// TwinCAT 3 PLC project Testing
// ProgramVersion: 3.1.4026.13
// libraries:
//   Tc2_Standard, * (Beckhoff Automation GmbH)
//   Tc2_System, * (Beckhoff Automation GmbH)
//   Tc3_Component, * (Zerlauth)
//   Tc3_Module, * (Beckhoff Automation GmbH)
//   Tc3_UnitTest, * (Zerlauth)
// project tree:
//   / PlcTask.TcTTO
//   POUs/ MAIN.TcPOU
//   Tests/ FB_ListComponentTests.TcPOU, FB_ListObjectTests.TcPOU, FB_ListStringTests.TcPOU, FB_MembersTests.TcPOU, FB_ComponentTests.TcPOU
// (motion and I/O tree: see PLC project development)
// real-time tasks:
//   TASK PlcTask: cycle T#500ms, priority 21, ADS port 351
//   TASK UnitTestTask: cycle T#1ms, priority 1, ADS port 350
// variable links:

CONFIGURATION Testing
    RESOURCE PLC ON TwinCAT3
        TASK PlcTask(INTERVAL := T#500ms, PRIORITY := 21);
        PROGRAM MAIN WITH PlcTask : MAIN;
    END_RESOURCE
END_CONFIGURATION

// ---- POUs/MAIN.TcPOU
PROGRAM MAIN
VAR
	bInitialise: 			BOOL:= TRUE;
	bExecute: 				BOOL;
	fbTestsuites:			FB_Testsuites;
	fbListObject:			FB_ListObjectTests;
	fbListComponent:		FB_ListComponentTests;
	fbListString:			FB_ListStringTests;
	fbMembers:				FB_MembersTests;
	fbComponentTests:		FB_ComponentTests;
END_VAR

IF bInitialise THEN
	bInitialise:= False;
	fbTestsuites.M_Add(fbListObject.fbTestsuite);
	fbTestsuites.M_Add(fbListComponent.fbTestsuite);
	fbTestsuites.M_Add(fbListString.fbTestsuite);
	fbTestsuites.M_Add(fbMembers.fbTestsuite);
	fbTestsuites.M_Add(fbComponentTests.fbTestsuite);
	fbTestsuites.P_Options.sFilePathName:= 'C:\report.xml';
END_IF

IF bExecute THEN
	bExecute:= fbTestsuites.M_Request(E_Base.Execute);
END_IF

fbTestsuites();


fbListObject();
fbListComponent();
fbListString();
fbMembers();
fbComponentTests();

END_PROGRAM

// ---- Tests/FB_ListObjectTests.TcPOU
FUNCTION_BLOCK FB_ListObjectTests EXTENDS 
VAR_INPUT
END_VAR
VAR_OUTPUT
	fbTestsuite:			FB_Testsuite;
END_VAR
VAR
	fbList:					Tc3_Component.FB_ListObject;
	fbObject:				Tc3_Component.FB_Object;
	iObject:				Tc3_Component.I_Object:= fbObject;
END_VAR

fbTestsuite.P_Property.M_Add('object', 'FB_ListObject');
fbTestsuite.P_Property.M_Add('name', 'Peter Zerlauth');

fbTestsuite();

CASE fbTestsuite.P_Testcase OF
	
	E_Testcase.Start:
		fbTestsuite.P_Assert.M_Equals_DINT(fbList.P_Length, 0, 'P_Length');
		fbTestsuite.M_Testcase('FB_ListObject', T#2S, 'fbList.P_Length', '', 10);	
		
	10:
		fbTestsuite.P_Assert.M_Equals_BOOL(fbList.M_Add(fbObject), TRUE, 'M_Add(fbObject)');
		fbTestsuite.M_Testcase('FB_ListObject', T#2S, 'fbList.M_Add(fbObject)', '', 20);
		
	20:
		fbTestsuite.P_Assert.M_Equals_DINT(fbList.P_Length, 1, 'P_Length');
		fbTestsuite.M_Testcase('FB_ListObject', T#2S, 'fbList.P_Length', '', 30);		
		
	30:
		fbTestsuite.P_Assert.M_Equals_DINT(fbList.M_Find(fbObject), 0, 'M_Find');
		fbTestsuite.M_Testcase('FB_ListObject', T#2S, 'fbList.M_Find(fbObject)', '', 40);
		
	40:

		fbTestsuite.P_Assert.M_Equals_BOOL(TRUE, __QUERYINTERFACE(fbList.M_Index(0), iObject), 'M_Index');
		fbTestsuite.M_Testcase('FB_ListObject', T#2S, 'fbList.M_Index(1)', '', 50);
		
	50:
		fbTestsuite.P_Assert.M_Equals_BOOL(fbList.M_Remove(fbObject), TRUE, 'M_Remove');
		fbTestsuite.M_Testcase('FB_ListObject', T#2S, 'fbList.M_Remove(fbObject', '', 60);		

	60:
		fbTestsuite.P_Assert.M_Equals_DINT(fbList.P_Length, 0, 'P_Length');
		fbTestsuite.M_Testcase('FB_ListObject', T#2S, 'fbList.P_Length', '', 70);
		
	70:
		fbTestsuite.P_Assert.M_Equals_BOOL(fbList.M_Add(fbObject), TRUE, 'M_Add(fbObject)');
		fbTestsuite.M_Testcase('FB_ListObject', T#2S, 'fbList.M_Add(fbObject)', '', 80);

	80:
		fbTestsuite.P_Assert.M_Equals_DINT(fbList.P_Length, 1, 'P_Length');
		fbTestsuite.M_Testcase('FB_ListObject', T#2S, 'fbList.P_Length', '', 90);
		
	90:
		fbTestsuite.P_Assert.M_Equals_BOOL(fbList.M_Clear(), TRUE, 'M_Clear()');
		fbTestsuite.M_Testcase('FB_ListObject', T#2S, 'fbList.M_Clear()', '', 100);		
	
	100:
		fbTestsuite.P_Assert.M_Equals_DINT(fbList.P_Length, 0, 'P_Length');
		fbTestsuite.M_Testcase('FB_ListObject', T#2S, 'fbList.P_Length', '', E_Testcase.Done);
		
	E_Testcase.Done:
		;
END_CASE

END_FUNCTION_BLOCK

// ---- Tests/FB_ListComponentTests.TcPOU
FUNCTION_BLOCK FB_ListComponentTests EXTENDS 
VAR_INPUT
END_VAR
VAR_OUTPUT
	fbTestsuite:			FB_Testsuite;
END_VAR
VAR
	fbList:					Tc3_Component.FB_ListComponent;
	fbObject:				Tc3_Component.FB_Component;
	iObject:				Tc3_Component.I_Component:= fbObject;
END_VAR

fbTestsuite.P_Property.M_Add('object', 'FB_ListComponent');
fbTestsuite.P_Property.M_Add('name', 'Peter Zerlauth');

fbTestsuite();

CASE fbTestsuite.P_Testcase OF
	
	E_Testcase.Start:
		fbTestsuite.P_Assert.M_Equals_DINT(fbList.P_Length, 0, 'P_Length');
		fbTestsuite.M_Testcase('FB_ListComponent', T#2S, 'fbList.P_Length', '', 10);	
		
	10:
		fbTestsuite.P_Assert.M_Equals_BOOL(fbList.M_Add(fbObject), TRUE, 'M_Add(fbObject)');
		fbTestsuite.M_Testcase('FB_ListComponent', T#2S, 'fbList.M_Add(fbObject)', '', 20);
		
	20:
		fbTestsuite.P_Assert.M_Equals_DINT(fbList.P_Length, 1, 'P_Length');
		fbTestsuite.M_Testcase('FB_ListComponent', T#2S, 'fbList.P_Length', '', 30);		
		
	30:
		fbTestsuite.P_Assert.M_Equals_DINT(fbList.M_Find(fbObject), 0, 'M_Find');
		fbTestsuite.M_Testcase('FB_ListComponent', T#2S, 'fbList.M_Find(fbObject)', '', 40);
		
	40:

		fbTestsuite.P_Assert.M_Equals_BOOL(TRUE, __QUERYINTERFACE(fbList.M_Index(0), iObject), 'M_Index');
		fbTestsuite.M_Testcase('FB_ListComponent', T#2S, 'fbList.M_Index(1)', '', 50);
		
	50:
		fbTestsuite.P_Assert.M_Equals_BOOL(fbList.M_Remove(fbObject), TRUE, 'M_Remove');
		fbTestsuite.M_Testcase('FB_ListComponent', T#2S, 'fbList.M_Remove(fbObject', '', 60);		

	60:
		fbTestsuite.P_Assert.M_Equals_DINT(fbList.P_Length, 0, 'P_Length');
		fbTestsuite.M_Testcase('FB_ListComponent', T#2S, 'fbList.P_Length', '', 70);
		
	70:
		fbTestsuite.P_Assert.M_Equals_BOOL(fbList.M_Add(fbObject), TRUE, 'M_Add(fbObject)');
		fbTestsuite.M_Testcase('FB_ListComponent', T#2S, 'fbList.M_Add(fbObject)', '', 80);

	80:
		fbTestsuite.P_Assert.M_Equals_DINT(fbList.P_Length, 1, 'P_Length');
		fbTestsuite.M_Testcase('FB_ListComponent', T#2S, 'fbList.P_Length', '', 90);
		
	90:
		fbTestsuite.P_Assert.M_Equals_BOOL(fbList.M_Clear(), TRUE, 'M_Clear()');
		fbTestsuite.M_Testcase('FB_ListComponent', T#2S, 'fbList.M_Clear()', '', 100);		
	
	100:
		fbTestsuite.P_Assert.M_Equals_DINT(fbList.P_Length, 0, 'P_Length');
		fbTestsuite.M_Testcase('FB_ListComponent', T#2S, 'fbList.P_Length', '', E_Testcase.Done);
		
	E_Testcase.Done:
		;
END_CASE

END_FUNCTION_BLOCK

// ---- Tests/FB_ListStringTests.TcPOU
FUNCTION_BLOCK FB_ListStringTests EXTENDS 
VAR_INPUT
END_VAR
VAR_OUTPUT
	fbTestsuite:			FB_Testsuite;
END_VAR
VAR
	fbList:					Tc3_Component.FB_ListString;
END_VAR

fbTestsuite.P_Property.M_Add('object', 'FB_ListString');
fbTestsuite.P_Property.M_Add('name', 'Peter Zerlauth');

fbTestsuite();

CASE fbTestsuite.P_Testcase OF
	
	E_Testcase.Start:
		fbTestsuite.P_Assert.M_Equals_DINT(fbList.P_Length, 0, 'P_Length');
		fbTestsuite.M_Testcase('FB_ListString', T#2S, 'fbList.P_Length', '', 10);	
		
	10:
		fbTestsuite.P_Assert.M_Equals_BOOL(fbList.M_Add('test'), TRUE, 'M_Add("test")');
		fbTestsuite.M_Testcase('FB_ListString', T#2S, 'fbList.M_Add(test)', '', 20);
		
	20:
		fbTestsuite.P_Assert.M_Equals_DINT(fbList.P_Length, 1, 'P_Length');
		fbTestsuite.M_Testcase('FB_ListString', T#2S, 'fbList.P_Length', '', 30);		
		
	30:
		fbTestsuite.P_Assert.M_Equals_DINT(fbList.M_Find('test'), 0, 'M_Find');
		fbTestsuite.M_Testcase('FB_ListString', T#2S, 'fbList.M_Find(test)', '', 40);
		
	40:

		fbTestsuite.P_Assert.M_Equals_BOOL(TRUE, fbList.M_Index(0) = 'test', 'M_Index');
		fbTestsuite.M_Testcase('FB_ListString', T#2S, 'fbList.M_Index(1)', '', 50);
		
	50:
		fbTestsuite.P_Assert.M_Equals_BOOL(fbList.M_Remove('test'), TRUE, 'M_Remove');
		fbTestsuite.M_Testcase('FB_ListString', T#2S, 'fbList.M_Remove(fbObject', '', 60);		

	60:
		fbTestsuite.P_Assert.M_Equals_DINT(fbList.P_Length, 0, 'P_Length');
		fbTestsuite.M_Testcase('FB_ListString', T#2S, 'fbList.P_Length', '', 70);
		
	70:
		fbTestsuite.P_Assert.M_Equals_BOOL(fbList.M_Add('test'), TRUE, 'M_Add(test)');
		fbTestsuite.M_Testcase('FB_ListString', T#2S, 'fbList.M_Add(test)', '', 80);

	80:
		fbTestsuite.P_Assert.M_Equals_DINT(fbList.P_Length, 1, 'P_Length');
		fbTestsuite.M_Testcase('FB_ListString', T#2S, 'fbList.P_Length', '', 90);
		
	90:
		fbTestsuite.P_Assert.M_Equals_BOOL(fbList.M_Clear(), TRUE, 'M_Clear()');
		fbTestsuite.M_Testcase('FB_ListString', T#2S, 'fbList.M_Clear()', '', 100);		
	
	100:
		fbTestsuite.P_Assert.M_Equals_DINT(fbList.P_Length, 0, 'P_Length');
		fbTestsuite.M_Testcase('FB_ListString', T#2S, 'fbList.P_Length', '', 110);
		
	110:	
		fbTestsuite.P_Assert.M_Equals_BOOL(fbList.M_Add(''), FALSE, 'M_Add("")');
		fbTestsuite.M_Testcase('FB_ListString', T#2S, 'fbList.M_Add(test)', '', 120);

	120:
		fbTestsuite.P_Assert.M_Equals_DINT(fbList.P_Length, 0, 'P_Length');
		fbTestsuite.M_Testcase('FB_ListString', T#2S, 'fbList.P_Length', '', E_Testcase.Done);	
		
		
	E_Testcase.Done:
		;
END_CASE

END_FUNCTION_BLOCK

// ---- Tests/FB_MembersTests.TcPOU
FUNCTION_BLOCK FB_MembersTests EXTENDS 
VAR_INPUT
END_VAR
VAR_OUTPUT
	fbTestsuite:			FB_Testsuite;
END_VAR
VAR
	fbList:					Tc3_Component.FB_Members;
	fbObject1:				Tc3_Component.FB_Component;
	fbObject2:				Tc3_Component.FB_Component;
END_VAR

fbTestsuite.P_Property.M_Add('object', 'FB_Members');
fbTestsuite.P_Property.M_Add('name', 'Peter Zerlauth');

fbTestsuite();

fbObject1();
fbObject2();

CASE fbTestsuite.P_Testcase OF
	
	E_Testcase.Start:
		fbList.M_Clear();
		fbTestsuite.P_Assert.M_Equals_DINT(fbList.P_Length, 0, 'P_Length');
		fbTestsuite.M_Testcase('FB_Members', T#2S, 'fbList.P_Length', '', 10);	
		
	10:
		fbTestsuite.P_Assert.M_Equals_BOOL(fbList.M_Add(fbObject1), TRUE, 'M_Add(fbObject1)');
		fbTestsuite.P_Assert.M_Equals_BOOL(fbList.M_Add(fbObject2), TRUE, 'M_Add(fbObject2)');
		fbTestsuite.P_Assert.M_Equals_DINT(fbList.P_Length, 2, 'P_Length');
		fbTestsuite.M_Testcase('FB_Members', T#2S, 'fbList.M_Add(fbObject)', '', 20);
		
	20:
		fbTestsuite.P_Assert.M_Equals_BOOL(fbList.M_Start(), 1, 'M_Start()');
		fbTestsuite.P_Assert.M_Equals_DINT(fbObject1.P_State, E_State.Execute, 'P_State');
		fbTestsuite.M_Testcase('FB_Members', T#2S, 'fbList.M_Start()', '', 30);		
		
	30:
		fbTestsuite.P_Assert.M_Equals_BOOL(fbList.M_Stop(), 1, 'M_Stop()');
		fbTestsuite.P_Assert.M_Equals_DINT(fbObject1.P_State, E_State.Stopped, 'P_State');
		fbTestsuite.M_Testcase('FB_Members', T#2S, 'fbList.M_Stop()', '', 40);
		
	40:

		fbTestsuite.P_Assert.M_Equals_BOOL(fbList.M_Reset(), 1, 'M_Reset()');
		fbTestsuite.P_Assert.M_Equals_DINT(fbObject1.P_State, E_State.Idle, 'P_State');
		fbTestsuite.M_Testcase('FB_Members', T#2S, 'fbList.M_Reset()', '', 50);
		
	50:
		fbTestsuite.P_Assert.M_Equals_BOOL(fbList.M_Start(), 1, 'M_Start()');
		fbTestsuite.P_Assert.M_Equals_DINT(fbObject1.P_State, E_State.Execute, 'P_State');
		fbTestsuite.M_Testcase('FB_Members', T#2S, 'fbList.M_Start()', '', 60);		

	60:
		fbTestsuite.P_Assert.M_Equals_BOOL(fbList.M_Abort(), 1, 'M_Abort()');
		fbTestsuite.P_Assert.M_Equals_DINT(fbObject1.P_State, E_State.Aborted, 'P_State');
		fbTestsuite.M_Testcase('FB_Members', T#2S, 'fbList.M_Abort()', '', 70);
		
	70:
		fbTestsuite.P_Assert.M_Equals_BOOL(fbList.M_Reset(), 1, 'M_Reset()');
		fbTestsuite.P_Assert.M_Equals_DINT(fbObject1.P_State, E_State.Idle, 'P_State');
		fbTestsuite.M_Testcase('FB_Members', T#2S, 'fbList.M_Reset()', '',E_Testcase.Done);
		
	E_Testcase.Done:
		;
END_CASE

END_FUNCTION_BLOCK

// ---- Tests/FB_ComponentTests.TcPOU
FUNCTION_BLOCK FB_ComponentTests
VAR_INPUT
END_VAR
VAR_OUTPUT
	fbTestsuite:			FB_Testsuite;
END_VAR
VAR
	fbComponent:				Tc3_Component.FB_Component;
END_VAR

fbTestsuite.P_Property.M_Add('object', 'FB_Component');
fbTestsuite.P_Property.M_Add('name', 'Peter Zerlauth');

fbTestsuite();

fbComponent();

CASE fbTestsuite.P_Testcase OF
	
	E_Testcase.Start:
		IF fbComponent.P_State = E_State.Aborted THEN
			fbComponent.M_Request(E_Request.Reset);
		ELSIF	fbComponent.P_State <> E_State.Idle THEN
			fbComponent.M_Request(E_Request.Abort);			
		END_IF

		fbTestsuite.P_Assert.M_Equals_STRING(TO_STRING(E_State.Idle), TO_STRING(fbComponent.P_State), 'P_State');
		fbTestsuite.M_Testcase('FB_Component', T#2S, 'fbComponent.M_Request(E_Request.Reset)', '', 10);	
		
	10:
		fbTestsuite.P_Assert.M_Equals_BOOL(TRUE, fbComponent.M_Request(E_Request.Start), 'M_Request(E_Request.Start)');	
		fbTestsuite.P_Assert.M_Equals_STRING(TO_STRING(E_State.Execute), TO_STRING(fbComponent.P_State), 'P_State');
		fbTestsuite.M_Testcase('FB_Component', T#2S, 'fbComponent.M_Request(E_Request.Reset)', '', 20);
		
	20:
		fbTestsuite.P_Assert.M_Equals_BOOL(TRUE, fbComponent.M_Request(E_Request.Abort), 'M_Request(E_Request.Abort)');	
		fbTestsuite.P_Assert.M_Equals_STRING(TO_STRING(E_State.Aborted), TO_STRING(fbComponent.P_State), 'P_State');
		fbTestsuite.M_Testcase('FB_Component', T#2S, 'fbComponent.M_Request(E_Request.Abort)', '', 30);

	30:
		fbTestsuite.P_Assert.M_Equals_BOOL(TRUE, fbComponent.M_Request(E_Request.Reset), 'M_Request(E_Request.Reset)');	
		fbTestsuite.P_Assert.M_Equals_STRING(TO_STRING(E_State.Idle), TO_STRING(fbComponent.P_State), 'P_State');
		fbTestsuite.M_Testcase('FB_Component', T#2S, 'fbComponent.M_Request(E_Request.Reset)', '', 40);

	40:
		fbTestsuite.P_Assert.M_Equals_BOOL(TRUE, fbComponent.M_Request(E_Request.Start), 'M_Request(E_Request.Start)');	
		fbTestsuite.P_Assert.M_Equals_STRING(TO_STRING(E_State.Execute), TO_STRING(fbComponent.P_State), 'P_State');
		fbTestsuite.M_Testcase('FB_Component', T#2S, 'fbComponent.M_Request(E_Request.Reset)', '', 50);
		
	50:
		fbTestsuite.P_Assert.M_Equals_BOOL(TRUE, fbComponent.M_Request(E_Request.Stop), 'M_Request(E_Request.Stop)');	
		fbTestsuite.P_Assert.M_Equals_STRING(TO_STRING(E_State.Stopped), TO_STRING(fbComponent.P_State), 'P_State');
		fbTestsuite.M_Testcase('FB_Component', T#2S, 'fbComponent.M_Request(E_Request.Stop)', '', 60);
		
	60:
		fbTestsuite.P_Assert.M_Equals_BOOL(TRUE, fbComponent.M_Request(E_Request.Reset), 'M_Request(E_Request.Reset)');	
		fbTestsuite.P_Assert.M_Equals_STRING(TO_STRING(E_State.Idle), TO_STRING(fbComponent.P_State), 'P_State');
		fbTestsuite.M_Testcase('FB_Component', T#2S, 'fbComponent.M_Request(E_Request.Reset)', '', 70);
		
	70:
		fbComponent.P_Event.M_Abort('Abort', 1);
		fbTestsuite.P_Assert.M_Equals_STRING(TO_STRING(E_State.Aborted), TO_STRING(fbComponent.P_State), 'P_State');
		fbTestsuite.M_Testcase('FB_Component', T#2S, 'fbComponent.P_Event.M_Abort(Abort, 1)', '', E_Testcase.Done);		
		
		
	E_Testcase.Done:
		;
END_CASE

END_FUNCTION_BLOCK
